(* IEC 61131-3 sources: RL_MAR/experiments/comparison/llm4plc/results/gpt-4o-mini_20260506_100619/20260506_101952, 4 files *)

(* ---- generated_code_iteration_0.st ---- *)
ructured-text
START_ST
FUNCTION_BLOCK FB_RealValueAdjuster
VAR_INPUT
    x_in : REAL; // Input variable of type REAL
END_VAR

VAR_OUTPUT
    x_out : REAL; // Output variable of type REAL
END_VAR

VAR
    x : REAL; // Internal variable to hold the adjusted value
    int_x : INT; // Internal variable to hold the integer conversion of x_in
END_VAR

// Initialize the output variable
x_out := 0.0; // Initialize the output variable

// Processing logic
// Check if x_in is exactly 0.0
IF x_in = 0.0 THEN
    x := x_in + 1.0; // Add 1.0 if input is 0.0
ELSE
    x := x_in + 1.0; // Add 1.0 if input is not 0.0
END_IF;

// Convert the real input to an integer
int_x := INT(x_in);

// Check if the integer conversion is not zero
IF int_x <> 0 THEN
    x := x + 1.0; // Add 1.0 to the adjusted value if int_x is not zero
END_IF;

// Assign the final adjusted value to the output variable
x_out := x;

END_FUNCTION_BLOCK
END_ST

(* ---- generated_code_iteration_1.st ---- *)
START_REASON
The errors in the original Structured Text (ST) code occurred due to the incorrect use of the "INT" keyword. In Structured Text, the "INT" type should not be used as a standalone statement; instead, it should be part of an assignment or conversion operation. The feedback indicated that the code failed the CODESYS compiler validation because of this issue. Additionally, the code structure and logic need to be maintained as a FUNCTION_BLOCK, and variable sections must be properly closed with "END_VAR".
END_REASON

START_ST
FUNCTION_BLOCK FB_RealValueAdjuster
VAR_INPUT
    x_in : REAL; // Input variable of type REAL
END_VAR

VAR_OUTPUT
    x_out : REAL; // Output variable of type REAL
END_VAR

VAR
    x : REAL; // Internal variable to hold the adjusted value
    int_x : INT; // Internal variable to hold the integer conversion of x_in
END_VAR

// Initialize the output variable
x_out := 0.0; // Initialize the output variable

// Processing logic
// Check if x_in is exactly 0.0
IF x_in = 0.0 THEN
    x := x_in + 1.0; // Add 1.0 if input is 0.0
ELSE
    x := x_in + 1.0; // Add 1.0 if input is not 0.0
END_IF;

// Convert the real input to an integer
int_x := INT(x_in); // Correctly assign the integer conversion of x_in

// Check if the integer conversion is not zero
IF int_x <> 0 THEN
    x := x + 1.0; // Add 1.0 to the adjusted value if int_x is not zero
END_IF;

// Assign the final adjusted value to the output variable
x_out := x;

END_FUNCTION_BLOCK
END_ST

(* ---- generated_code_iteration_2.st ---- *)
START_REASON
The errors in the original Structured Text (ST) code occurred due to the incorrect use of the "INT" keyword. In Structured Text, the "INT" type should not be used as a standalone statement; instead, it should be part of an assignment or conversion operation. The feedback indicated that the code failed the CODESYS compiler validation because of this issue. Additionally, the code structure and logic need to be maintained as a FUNCTION_BLOCK, and variable sections must be properly closed with "END_VAR". The proper syntax for type conversion should be used to ensure the code compiles correctly.
END_REASON

START_ST
FUNCTION_BLOCK FB_RealValueAdjuster
VAR_INPUT
    x_in : REAL; // Input variable of type REAL
END_VAR

VAR_OUTPUT
    x_out : REAL; // Output variable of type REAL
END_VAR

VAR
    x : REAL; // Internal variable to hold the adjusted value
    int_x : INT; // Internal variable to hold the integer conversion of x_in
END_VAR

// Initialize the output variable
x_out := 0.0; // Initialize the output variable

// Processing logic
// Check if x_in is exactly 0.0
IF x_in = 0.0 THEN
    x := x_in + 1.0; // Add 1.0 if input is 0.0
ELSE
    x := x_in + 1.0; // Add 1.0 if input is not 0.0
END_IF;

// Convert the real input to an integer
int_x := TRUNC(x_in); // Correctly assign the integer conversion of x_in

// Check if the integer conversion is not zero
IF int_x <> 0 THEN
    x := x + 1.0; // Add 1.0 to the adjusted value if int_x is not zero
END_IF;

// Assign the final adjusted value to the output variable
x_out := x;

END_FUNCTION_BLOCK
END_ST

(* ---- generated_code_iteration_3.st ---- *)
START_REASON
The errors in the original Structured Text (ST) code occurred due to the incorrect handling of data types, specifically the conversion of a REAL type to an INT type. The feedback indicates that there was an attempt to convert a DINT type to an INT type, which is not allowed. This suggests that the TRUNC function may be returning a DINT instead of an INT. To fix this, I will ensure that the conversion is handled properly and that the variable types are consistent throughout the code. Additionally, I will maintain the structure of the FUNCTION_BLOCK and ensure all variable sections are properly closed with "END_VAR".
END_REASON

START_ST
FUNCTION_BLOCK FB_RealValueAdjuster
VAR_INPUT
    x_in : REAL; // Input variable of type REAL
END_VAR

VAR_OUTPUT
    x_out : REAL; // Output variable of type REAL
END_VAR

VAR
    x : REAL; // Internal variable to hold the adjusted value
    int_x : INT; // Internal variable to hold the integer conversion of x_in
END_VAR

// Initialize the output variable
x_out := 0.0; // Initialize the output variable

// Processing logic
// Check if x_in is exactly 0.0
IF x_in = 0.0 THEN
    x := x_in + 1.0; // Add 1.0 if input is 0.0
ELSE
    x := x_in + 1.0; // Add 1.0 if input is not 0.0
END_IF;

// Convert the real input to an integer
int_x := INT(TRUNC(x_in)); // Correctly assign the integer conversion of x_in

// Check if the integer conversion is not zero
IF int_x <> 0 THEN
    x := x + 1.0; // Add 1.0 to the adjusted value if int_x is not zero
END_IF;

// Assign the final adjusted value to the output variable
x_out := x;

END_FUNCTION_BLOCK
END_ST
